FUNCTION Convert_SINT_TO_BYTE : BOOL
VAR_INPUT
	in : SINT;
	out : REFERENCE TO BYTE;
END_VAR
VAR
	converted : BYTE;
END_VAR

converted := SINT_TO_BYTE(in);

IF (BYTE_TO_SINT(converted) <> in) THEN
	RETURN;
END_IF

out := converted;
Convert_SINT_TO_BYTE := TRUE;

END_FUNCTION

(* stored: Version 1.1.0.1, ProductVersion 3.1.4024.12
   POU Convert_SINT_TO_BYTE: Id {ba385739-9e17-4302-9aee-0b7d4e3a6cc3}, SpecialFunc None *)
